Fanuc TP program (LS listing): PICK.LS

/PROG  PICK
/ATTR
OWNER		= MNEDITOR;
COMMENT		= "Pick            ";
PROG_SIZE	= 696;
CREATE		= DATE 26-09-18  TIME 12:01:46;
MODIFIED	= DATE 26-09-18  TIME 12:01:46;
FILE_NAME	= ;
VERSION		= 0;
LINE_COUNT	= 9;
MEMORY_SIZE	= 1032;
PROTECT		= READ_WRITE;
TCD:  STACK_SIZE	= 0,
      TASK_PRIORITY	= 50,
      TIME_SLICE	= 0,
      BUSY_LAMP_OFF	= 0,
      ABORT_REQUEST	= 0,
      PAUSE_REQUEST	= 0;
DEFAULT_GROUP	= 1,*,*,*,*;
CONTROL_CODE	= 00000000 00000000;
LOCAL_REGISTERS	= 0,0,0;
/MN
   1:  !RAPID PickAndPlace.Pick ;
   2:  ! approach, grip, retract ;
   3:  UFRAME_NUM=0 ;
   4:  UTOOL_NUM=2 ;
   5:J P[1] 50% CNT20    ;
   6:L P[2] 200mm/sec FINE    ;
   7:  DO[1]=ON ;
   8:  WAIT    .30(sec) ;
   9:L P[1] 500mm/sec CNT10    ;
/POS
P[1]{
   GP1:
	UF : 0, UT : 2,		CONFIG : 'N U T, 0, 0, 0',
	X =   812.350  mm,	Y =  -245.100  mm,	Z =   405.000  mm,
	W =  -179.293 deg,	P =     0.000 deg,	R =   -90.000 deg
};
P[2]{
   GP1:
	UF : 0, UT : 2,		CONFIG : 'N U T, 0, 0, 0',
	X =   812.350  mm,	Y =  -245.100  mm,	Z =   305.000  mm,
	W =  -179.293 deg,	P =     0.000 deg,	R =   -90.000 deg
};
/END
